TYPE ST_Contactor_Status :
    STRUCT
        Extended   : BOOL;
        Retracted  : BOOL;
        Extending  : BOOL;
        Retracting : BOOL;
    END_STRUCT
END_TYPE

(* stored: Version 1.1.0.1, ProductVersion 3.1.4024.15
   DUT ST_Contactor_Status: Id {657e4614-e956-4472-978d-dd9d151c2bc2} *)
